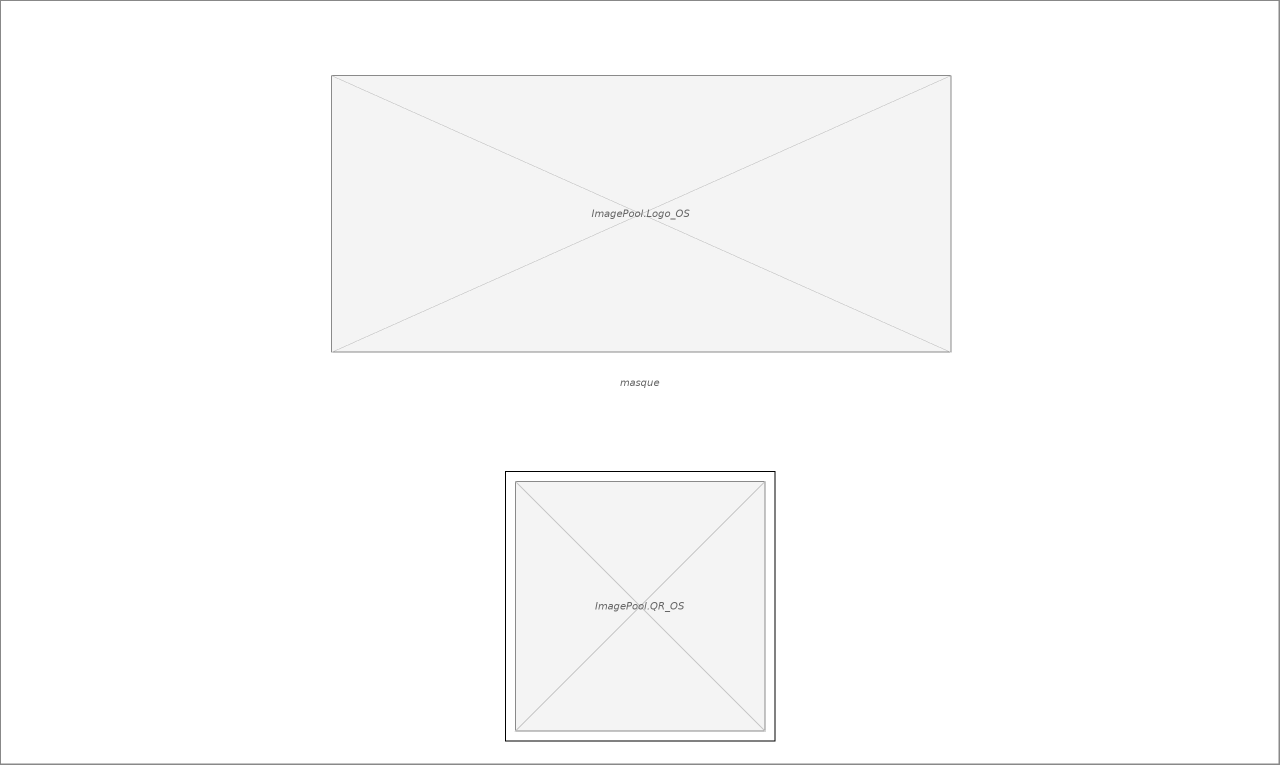
VISUALIZATION Accueil  // 1280x765
    Frame (0,0 1280x765)
        shows masque()
    RoundedRectangle (0,383 1280x80), "Phone : +33 (0)4 93 77 79 74"
    RoundedRectangle (0,303 1280x80), "Mail : Smartbooth@osmose06.com"
    RoundedRectangle (340,153 600x126)
    Image (331,75 620x277), image: ImagePool.Logo_OS
    Rectangle (0,128 1278x633)
        OnMouseDown: change screen: menu
    Group (505,471 270x270)
        RoundedRectangle (0,0 270x270)
        Image (10,10 250x250), image: ImagePool.QR_OS
END_VISUALIZATION

(* stored: Version 1.1.0.1, ProductVersion 3.1.4024.15
   Visu Accueil: Id {7446499b-a33a-47fc-b8d8-3ead0c4d6a46} *)
